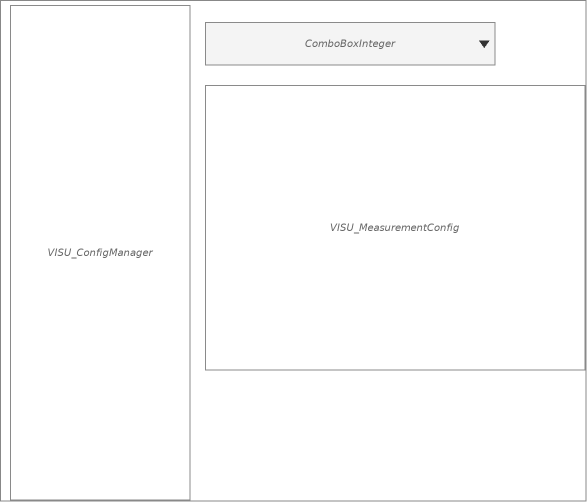
VISUALIZATION VISU_TelemetryConfig  // 587x502
VAR_IN_OUT
    editable : TelemetryConfig;
	active : TelemetryConfig;
    mgr : ConfigManager;
    mgrWidget : ConfigManagerWidget;
    telemetryWidget : TelemetryWidget;
END_VAR
    Frame (10,5 180x495)
        shows VISU_ConfigManager(mgr := mgr, widget := mgrWidget)
    ComboBoxInteger (205,22 290x43), variable: telemetryWidget.activeConfigTab, text list: 'TelemetryConfigTextList'
    Frame (205,85 380x285), frame switch variable: telemetryWidget.activeConfigTab
        shows VISU_MeasurementConfig(active := active.temperatures.m1, editable := editable.temperatures.m1)
        shows VISU_MeasurementConfig(active := active.temperatures.mirrorCell, editable := editable.temperatures.mirrorCell)
        shows VISU_MeasurementConfig(active := active.temperatures.m2, editable := editable.temperatures.m2)
        shows VISU_MeasurementConfig(active := active.temperatures.m2Electronics, editable := editable.temperatures.m2Electronics)
        shows VISU_MeasurementConfig(active := active.temperatures.topTube, editable := editable.temperatures.topTube)
        shows VISU_MeasurementConfig(active := active.temperatures.centreTube, editable := editable.temperatures.centreTube)
        shows VISU_MeasurementConfig(active := active.temperatures.fork, editable := editable.temperatures.fork)
        shows VISU_MeasurementConfig(active := active.temperatures.nasmythAir, editable := editable.temperatures.nasmythAir)
        shows VISU_MeasurementConfig(active := active.temperatures.rem, editable := editable.temperatures.rem)
        shows VISU_MeasurementConfig(active := active.temperatures.rpm, editable := editable.temperatures.rpm)
        shows VISU_MeasurementConfig(active := active.temperatures.hermesTelescopeAdapter, editable := editable.temperatures.hermesTelescopeAdapter)
        shows VISU_MeasurementConfig(active := active.temperatures.topAir, editable := editable.temperatures.topAir)
        shows VISU_MeasurementConfig(active := active.temperatures.insideTube, editable := editable.temperatures.insideTube)
        shows VISU_MeasurementConfig(active := active.relativeHumidities.topAir, editable := editable.relativeHumidities.topAir)
        shows VISU_MeasurementConfig(active := active.relativeHumidities.insideTube, editable := editable.relativeHumidities.insideTube)
        shows VISU_MeasurementConfig(active := active.dewpoints.topAir, editable := editable.dewpoints.topAir)
        shows VISU_MeasurementConfig(active := active.dewpoints.insideTube, editable := editable.dewpoints.insideTube)
        shows VISU_MeasurementConfig(active := active.accelerometers.tube.x, editable := editable.accelerometers.tube.x)
        shows VISU_MeasurementConfig(active := active.accelerometers.tube.y, editable := editable.accelerometers.tube.y)
END_VISUALIZATION

(* stored: Version 1.1.0.1, ProductVersion 3.1.4019.2
   Visu VISU_TelemetryConfig: Id {c0cc9b15-9816-4a52-9b85-58bc2eb8853c} *)
